{attribute 'linkalways'} 
{attribute 'no_explicit_call' := 'This FB is a CLASS and must be accessed using methods or properties'}
{attribute 'enable_dynamic_creation'}
FUNCTION_BLOCK FINAL GE_LWORD EXTENDS Node
VAR
	in1 : _LWORD(0);
	in2 : _LWORD(0);
	out : _BOOL(FALSE);
END_VAR

METHOD PUBLIC Clone : I_Node
VAR
	pNode : POINTER TO GE_LWORD;
END_VAR
pNode := __NEW(GE_LWORD);
Clone := pNode^;
END_METHOD

METHOD FB_init : BOOL
VAR_INPUT
	bInitRetains : BOOL; // if TRUE, the retain variables are initialized (warm start / cold start)
	bInCopyCode : BOOL;  // if TRUE, the instance afterwards gets moved into the copy code (online change)
END_VAR
AddInput('in1',THIS^.in1);
AddInput('in2',THIS^.in2);
AddOutput('out', THIS^.out);
END_METHOD

METHOD PROTECTED OnExecute
VAR
END_VAR
out.Value := in1.Value >= in2.Value;
END_METHOD

END_FUNCTION_BLOCK

(* stored: Version 1.1.0.1, ProductVersion 3.1.4024.15
   POU GE_LWORD: Id {597d2905-fe05-42da-9e09-872ec280df66}, SpecialFunc None
   Folder Constructor: Id {fc277b88-51e9-432f-8fb0-db2566938cd3}
   Method Clone: Id {35048a71-82fe-4e1c-9b91-af4606356fca}
   Method FB_init: Id {39d1dfd0-f615-4105-aecc-68d204eac2c1}
   Method OnExecute: Id {896e6bb6-0f0b-48b4-b62d-81a71c8b8062} *)
